PROGRAM main
VAR_INPUT
	X0 : bool;
	X1 : bool;
END_VAR

VAR_OUTPUT
	Y0 : bool;
END_VAR

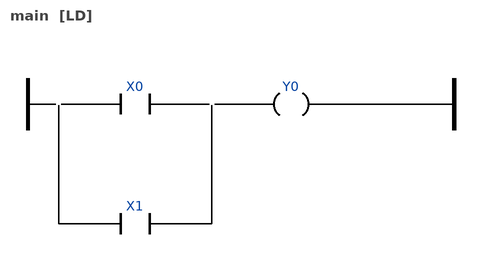
(* LD diagram, written out as Structured Text *)
Y0 := X0 OR X1;
END_PROGRAM
